LAYER IOs
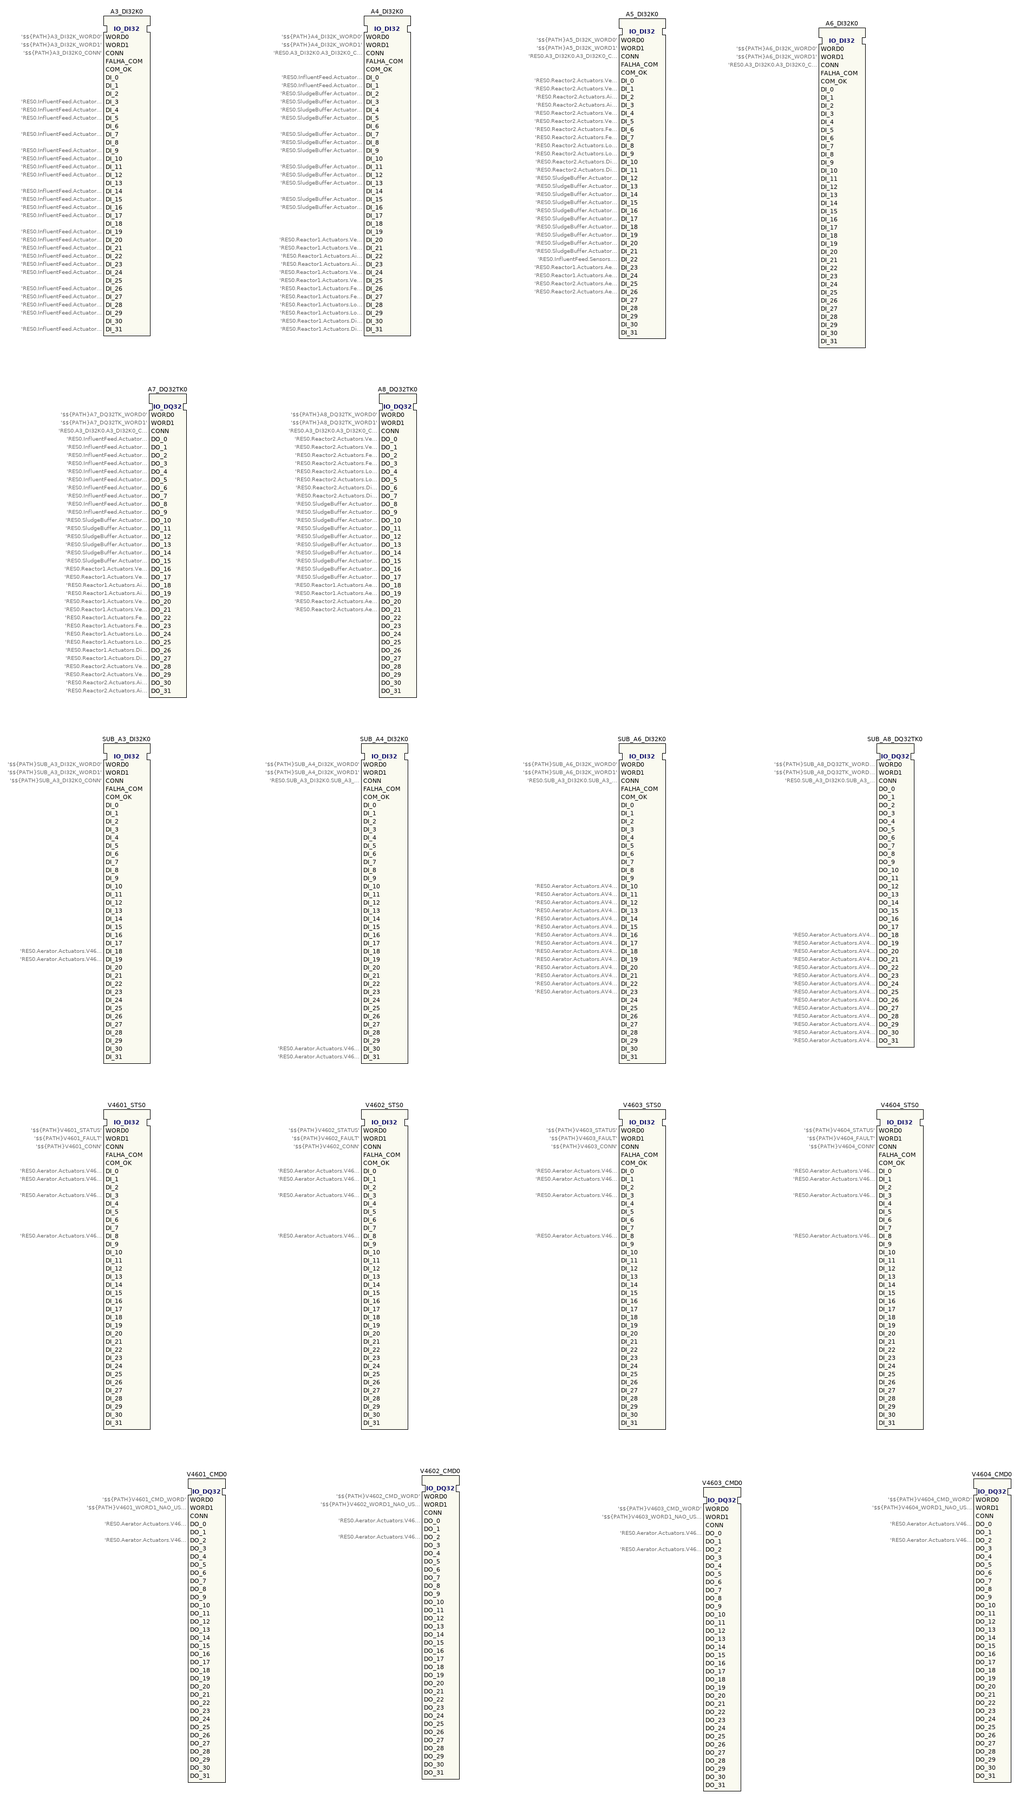
  FBS
    A3_DI32K0 : IO_DI32(WORD0 := '$${PATH}A3_DI32K_WORD0', WORD1 := '$${PATH}A3_DI32K_WORD1', DI_3 := 'RES0.InfluentFeed.Actuators.FeedReactorPump01.LocalPanel.SafetySwitchOff', DI_4 := 'RES0.InfluentFeed.Actuators.FeedReactorPump02.LocalPanel.SafetySwitchOff', DI_5 := 'RES0.InfluentFeed.Actuators.FeedReactorPump03.LocalPanel.SafetySwitchOff', DI_7 := 'RES0.InfluentFeed.Actuators.FeedReactorPump01.LocalPanel.RemoteSelect', DI_9 := 'RES0.InfluentFeed.Actuators.FeedReactorPump01.fbFwd.DIn', DI_10 := 'RES0.InfluentFeed.Actuators.FeedReactorPump01.LocalPanel.ElectricCircuitFail', DI_11 := 'RES0.InfluentFeed.Actuators.FeedReactorPump01.LocalPanel.MoistureDetectionPumpMS', DI_12 := 'RES0.InfluentFeed.Actuators.FeedReactorPump02.LocalPanel.RemoteSelect', DI_14 := 'RES0.InfluentFeed.Actuators.FeedReactorPump02.fbFwd.DIn', DI_15 := 'RES0.InfluentFeed.Actuators.FeedReactorPump02.LocalPanel.ElectricCircuitFail', DI_16 := 'RES0.InfluentFeed.Actuators.FeedReactorPump02.LocalPanel.MoistureDetectionPumpMS', DI_17 := 'RES0.InfluentFeed.Actuators.FeedReactorPump03.LocalPanel.RemoteSelect', DI_19 := 'RES0.InfluentFeed.Actuators.FeedReactorPump03.fbFwd.DIn', DI_20 := 'RES0.InfluentFeed.Actuators.FeedReactorPump03.LocalPanel.ElectricCircuitFail', DI_21 := 'RES0.InfluentFeed.Actuators.FeedReactorPump03.LocalPanel.MoistureDetectionPumpMS', DI_22 := 'RES0.InfluentFeed.Actuators.Mixer01.LocalPanel.PowerFb', DI_23 := 'RES0.InfluentFeed.Actuators.Mixer02.LocalPanel.PowerFb', DI_24 := 'RES0.InfluentFeed.Actuators.Mixer01.LocalPanel.RemoteSelect', DI_26 := 'RES0.InfluentFeed.Actuators.Mixer01.fbFwd.DIn', DI_27 := 'RES0.InfluentFeed.Actuators.Mixer01.LocalPanel.ElectricCircuitFail', DI_28 := 'RES0.InfluentFeed.Actuators.Mixer01.LocalPanel.MoistureDetectionPumpMS', DI_29 := 'RES0.InfluentFeed.Actuators.Mixer02.LocalPanel.RemoteSelect', DI_31 := 'RES0.InfluentFeed.Actuators.Mixer02.fbFwd.DIn', CONN := '$${PATH}A3_DI32K0_CONN');
    A4_DI32K0 : IO_DI32(WORD0 := '$${PATH}A4_DI32K_WORD0', WORD1 := '$${PATH}A4_DI32K_WORD1', DI_0 := 'RES0.InfluentFeed.Actuators.Mixer02.LocalPanel.ElectricCircuitFail', DI_1 := 'RES0.InfluentFeed.Actuators.Mixer02.LocalPanel.MoistureDetectionPumpMS', DI_2 := 'RES0.SludgeBuffer.Actuators.Pump1.LocalPanel.PowerFb', DI_3 := 'RES0.SludgeBuffer.Actuators.Pump2.LocalPanel.PowerFb', DI_4 := 'RES0.SludgeBuffer.Actuators.Pump3.LocalPanel.PowerFb', DI_5 := 'RES0.SludgeBuffer.Actuators.Pump1.LocalPanel.RemoteSelect', DI_7 := 'RES0.SludgeBuffer.Actuators.Pump1.fbFwd.DIn', DI_8 := 'RES0.SludgeBuffer.Actuators.Pump1.LocalPanel.ElectricCircuitFail', DI_9 := 'RES0.SludgeBuffer.Actuators.Pump2.LocalPanel.RemoteSelect', DI_11 := 'RES0.SludgeBuffer.Actuators.Pump2.fbFwd.DIn', DI_12 := 'RES0.SludgeBuffer.Actuators.Pump2.LocalPanel.ElectricCircuitFail', DI_13 := 'RES0.SludgeBuffer.Actuators.Pump3.LocalPanel.RemoteSelect', DI_15 := 'RES0.SludgeBuffer.Actuators.Pump3.fbFwd.DIn', DI_16 := 'RES0.SludgeBuffer.Actuators.Pump3.LocalPanel.ElectricCircuitFail', DI_20 := 'RES0.Reactor1.Actuators.VentAerationGridValve_AV4x107.fbOpen.DIn', DI_21 := 'RES0.Reactor1.Actuators.VentAerationGridValve_AV4x107.fbClose.DIn', DI_22 := 'RES0.Reactor1.Actuators.AirFillValveSludgeDischarge_AV4x171.fbOpen.DIn', DI_23 := 'RES0.Reactor1.Actuators.AirFillValveSludgeDischarge_AV4x171.fbClose.DIn', DI_24 := 'RES0.Reactor1.Actuators.VentSludgeGridValve_AV4x172.fbOpen.DIn', DI_25 := 'RES0.Reactor1.Actuators.VentSludgeGridValve_AV4x172.fbClose.DIn', DI_26 := 'RES0.Reactor1.Actuators.FeedValve_AV4x101.fbOpen.DIn', DI_27 := 'RES0.Reactor1.Actuators.FeedValve_AV4x101.fbClose.DIn', DI_28 := 'RES0.Reactor1.Actuators.LowerLevelValve_AV4x102.fbOpen.DIn', DI_29 := 'RES0.Reactor1.Actuators.LowerLevelValve_AV4x102.fbClose.DIn', DI_30 := 'RES0.Reactor1.Actuators.DischargeValve_AV4x103.fbOpen.DIn', DI_31 := 'RES0.Reactor1.Actuators.DischargeValve_AV4x103.fbClose.DIn', CONN := 'RES0.A3_DI32K0.A3_DI32K0_CONN');
    A5_DI32K0 : IO_DI32(WORD0 := '$${PATH}A5_DI32K_WORD0', WORD1 := '$${PATH}A5_DI32K_WORD1', DI_0 := 'RES0.Reactor2.Actuators.VentAerationGridValve_AV4x107.fbOpen.DIn', DI_1 := 'RES0.Reactor2.Actuators.VentAerationGridValve_AV4x107.fbClose.DIn', DI_2 := 'RES0.Reactor2.Actuators.AirFillValveSludgeDischarge_AV4x171.fbOpen.DIn', DI_3 := 'RES0.Reactor2.Actuators.AirFillValveSludgeDischarge_AV4x171.fbClose.DIn', DI_4 := 'RES0.Reactor2.Actuators.VentSludgeGridValve_AV4x172.fbOpen.DIn', DI_5 := 'RES0.Reactor2.Actuators.VentSludgeGridValve_AV4x172.fbClose.DIn', DI_6 := 'RES0.Reactor2.Actuators.FeedValve_AV4x101.fbOpen.DIn', DI_7 := 'RES0.Reactor2.Actuators.FeedValve_AV4x101.fbClose.DIn', DI_8 := 'RES0.Reactor2.Actuators.LowerLevelValve_AV4x102.fbOpen.DIn', DI_9 := 'RES0.Reactor2.Actuators.LowerLevelValve_AV4x102.fbClose.DIn', DI_10 := 'RES0.Reactor2.Actuators.DischargeValve_AV4x103.fbOpen.DIn', DI_11 := 'RES0.Reactor2.Actuators.DischargeValve_AV4x103.fbClose.DIn', DI_14 := 'RES0.SludgeBuffer.Actuators.ValveBuffer.fbOpen.DIn', DI_15 := 'RES0.SludgeBuffer.Actuators.ValveBuffer.fbClose.DIn', DI_16 := 'RES0.SludgeBuffer.Actuators.ValveInfeed.fbOpen.DIn', DI_17 := 'RES0.SludgeBuffer.Actuators.ValveInfeed.fbClose.DIn', DI_22 := 'RES0.InfluentFeed.Sensors.LevelSwitchInfluentBuffer.pv.DIn', DI_23 := 'RES0.Reactor1.Actuators.AerationBlockValve_AV4x170.fbOpen.DIn', DI_24 := 'RES0.Reactor1.Actuators.AerationBlockValve_AV4x170.fbClose.DIn', DI_25 := 'RES0.Reactor2.Actuators.AerationBlockValve_AV4x170.fbOpen.DIn', DI_26 := 'RES0.Reactor2.Actuators.AerationBlockValve_AV4x170.fbClose.DIn', CONN := 'RES0.A3_DI32K0.A3_DI32K0_CONN', DI_12 := 'RES0.SludgeBuffer.Actuators.ValveSupernatantReturn.fbOpen.DIn', DI_13 := 'RES0.SludgeBuffer.Actuators.ValveSupernatantReturn.fbClose.DIn', DI_18 := 'RES0.SludgeBuffer.Actuators.ValveTank2.fbOpen.DIn', DI_19 := 'RES0.SludgeBuffer.Actuators.ValveTank2.fbClose.DIn', DI_20 := 'RES0.SludgeBuffer.Actuators.ValveTank1.fbOpen.DIn', DI_21 := 'RES0.SludgeBuffer.Actuators.ValveTank1.fbClose.DIn');
    A6_DI32K0 : IO_DI32(WORD0 := '$${PATH}A6_DI32K_WORD0', WORD1 := '$${PATH}A6_DI32K_WORD1', CONN := 'RES0.A3_DI32K0.A3_DI32K0_CONN');
    A7_DQ32TK0 : IO_DQ32(WORD0 := '$${PATH}A7_DQ32TK_WORD0', WORD1 := '$${PATH}A7_DQ32TK_WORD1', DO_0 := 'RES0.InfluentFeed.Actuators.FeedReactorPump01.cmdFwd.DOut', DO_1 := 'RES0.InfluentFeed.Actuators.FeedReactorPump01.LocalPanel.ResetError_ATV', DO_2 := 'RES0.InfluentFeed.Actuators.FeedReactorPump02.cmdFwd.DOut', DO_3 := 'RES0.InfluentFeed.Actuators.FeedReactorPump02.LocalPanel.ResetError_ATV', DO_4 := 'RES0.InfluentFeed.Actuators.FeedReactorPump03.cmdFwd.DOut', DO_5 := 'RES0.InfluentFeed.Actuators.FeedReactorPump03.LocalPanel.ResetError_ATV', DO_6 := 'RES0.InfluentFeed.Actuators.Mixer01.cmdFwd.DOut', DO_7 := 'RES0.InfluentFeed.Actuators.Mixer01.LocalPanel.ResetError_ATV', DO_8 := 'RES0.InfluentFeed.Actuators.Mixer02.cmdFwd.DOut', DO_9 := 'RES0.InfluentFeed.Actuators.Mixer02.LocalPanel.ResetError_ATV', DO_10 := 'RES0.SludgeBuffer.Actuators.Pump1.cmdFwd.DOut', DO_11 := 'RES0.SludgeBuffer.Actuators.Pump1.LocalPanel.ResetError_ATV', DO_12 := 'RES0.SludgeBuffer.Actuators.Pump2.cmdFwd.DOut', DO_13 := 'RES0.SludgeBuffer.Actuators.Pump2.LocalPanel.ResetError_ATV', DO_14 := 'RES0.SludgeBuffer.Actuators.Pump3.cmdFwd.DOut', DO_15 := 'RES0.SludgeBuffer.Actuators.Pump3.LocalPanel.ResetError_ATV', DO_16 := 'RES0.Reactor1.Actuators.VentAerationGridValve_AV4x107.cmdOpen.DOut', DO_17 := 'RES0.Reactor1.Actuators.VentAerationGridValve_AV4x107.cmdClose.DOut', DO_18 := 'RES0.Reactor1.Actuators.AirFillValveSludgeDischarge_AV4x171.cmdOpen.DOut', DO_19 := 'RES0.Reactor1.Actuators.AirFillValveSludgeDischarge_AV4x171.cmdClose.DOut', DO_20 := 'RES0.Reactor1.Actuators.VentSludgeGridValve_AV4x172.cmdOpen.DOut', DO_21 := 'RES0.Reactor1.Actuators.VentSludgeGridValve_AV4x172.cmdClose.DOut', DO_22 := 'RES0.Reactor1.Actuators.FeedValve_AV4x101.cmdOpen.DOut', DO_23 := 'RES0.Reactor1.Actuators.FeedValve_AV4x101.cmdClose.DOut', DO_24 := 'RES0.Reactor1.Actuators.LowerLevelValve_AV4x102.cmdOpen.DOut', DO_25 := 'RES0.Reactor1.Actuators.LowerLevelValve_AV4x102.cmdClose.DOut', DO_26 := 'RES0.Reactor1.Actuators.DischargeValve_AV4x103.cmdOpen.DOut', DO_27 := 'RES0.Reactor1.Actuators.DischargeValve_AV4x103.cmdClose.DOut', DO_28 := 'RES0.Reactor2.Actuators.VentAerationGridValve_AV4x107.cmdOpen.DOut', DO_29 := 'RES0.Reactor2.Actuators.VentAerationGridValve_AV4x107.cmdClose.DOut', DO_30 := 'RES0.Reactor2.Actuators.AirFillValveSludgeDischarge_AV4x171.cmdOpen.DOut', DO_31 := 'RES0.Reactor2.Actuators.AirFillValveSludgeDischarge_AV4x171.cmdClose.DOut', CONN := 'RES0.A3_DI32K0.A3_DI32K0_CONN');
    A8_DQ32TK0 : IO_DQ32(WORD0 := '$${PATH}A8_DQ32TK_WORD0', WORD1 := '$${PATH}A8_DQ32TK_WORD1', DO_0 := 'RES0.Reactor2.Actuators.VentSludgeGridValve_AV4x172.cmdOpen.DOut', DO_1 := 'RES0.Reactor2.Actuators.VentSludgeGridValve_AV4x172.cmdClose.DOut', DO_2 := 'RES0.Reactor2.Actuators.FeedValve_AV4x101.cmdOpen.DOut', DO_3 := 'RES0.Reactor2.Actuators.FeedValve_AV4x101.cmdClose.DOut', DO_4 := 'RES0.Reactor2.Actuators.LowerLevelValve_AV4x102.cmdOpen.DOut', DO_5 := 'RES0.Reactor2.Actuators.LowerLevelValve_AV4x102.cmdClose.DOut', DO_6 := 'RES0.Reactor2.Actuators.DischargeValve_AV4x103.cmdOpen.DOut', DO_7 := 'RES0.Reactor2.Actuators.DischargeValve_AV4x103.cmdClose.DOut', DO_10 := 'RES0.SludgeBuffer.Actuators.ValveBuffer.cmdOpen.DOut', DO_11 := 'RES0.SludgeBuffer.Actuators.ValveBuffer.cmdClose.DOut', DO_12 := 'RES0.SludgeBuffer.Actuators.ValveInfeed.cmdOpen.DOut', DO_13 := 'RES0.SludgeBuffer.Actuators.ValveInfeed.cmdClose.DOut', DO_18 := 'RES0.Reactor1.Actuators.AerationBlockValve_AV4x170.cmdOpen.DOut', DO_19 := 'RES0.Reactor1.Actuators.AerationBlockValve_AV4x170.cmdClose.DOut', DO_20 := 'RES0.Reactor2.Actuators.AerationBlockValve_AV4x170.cmdOpen.DOut', DO_21 := 'RES0.Reactor2.Actuators.AerationBlockValve_AV4x170.cmdClose.DOut', CONN := 'RES0.A3_DI32K0.A3_DI32K0_CONN', DO_8 := 'RES0.SludgeBuffer.Actuators.ValveSupernatantReturn.cmdOpen.DOut', DO_9 := 'RES0.SludgeBuffer.Actuators.ValveSupernatantReturn.cmdClose.DOut', DO_17 := 'RES0.SludgeBuffer.Actuators.ValveTank1.cmdClose.DOut', DO_16 := 'RES0.SludgeBuffer.Actuators.ValveTank1.cmdOpen.DOut', DO_14 := 'RES0.SludgeBuffer.Actuators.ValveTank2.cmdOpen.DOut', DO_15 := 'RES0.SludgeBuffer.Actuators.ValveTank2.cmdClose.DOut');
    SUB_A3_DI32K0 : IO_DI32(WORD0 := '$${PATH}SUB_A3_DI32K_WORD0', WORD1 := '$${PATH}SUB_A3_DI32K_WORD1', DI_18 := 'RES0.Aerator.Actuators.V4603.LocalPanel.PowerFb', DI_19 := 'RES0.Aerator.Actuators.V4604.LocalPanel.PowerFb', CONN := '$${PATH}SUB_A3_DI32K0_CONN');
    SUB_A4_DI32K0 : IO_DI32(WORD0 := '$${PATH}SUB_A4_DI32K_WORD0', WORD1 := '$${PATH}SUB_A4_DI32K_WORD1', DI_30 := 'RES0.Aerator.Actuators.V4601.LocalPanel.PowerFb', DI_31 := 'RES0.Aerator.Actuators.V4602.LocalPanel.PowerFb', CONN := 'RES0.SUB_A3_DI32K0.SUB_A3_DI32K0_CONN');
    SUB_A6_DI32K0 : IO_DI32(WORD0 := '$${PATH}SUB_A6_DI32K_WORD0', WORD1 := '$${PATH}SUB_A6_DI32K_WORD1', DI_10 := 'RES0.Aerator.Actuators.AV46_001.fbOpen.DIn', DI_11 := 'RES0.Aerator.Actuators.AV46_001.fbClose.DIn', DI_12 := 'RES0.Aerator.Actuators.AV46_002.fbOpen.DIn', DI_13 := 'RES0.Aerator.Actuators.AV46_002.fbClose.DIn', DI_14 := 'RES0.Aerator.Actuators.AV46_003.fbOpen.DIn', DI_15 := 'RES0.Aerator.Actuators.AV46_003.fbClose.DIn', DI_16 := 'RES0.Aerator.Actuators.AV46_012.fbOpen.DIn', DI_17 := 'RES0.Aerator.Actuators.AV46_012.fbClose.DIn', DI_18 := 'RES0.Aerator.Actuators.AV46_022.fbOpen.DIn', DI_19 := 'RES0.Aerator.Actuators.AV46_022.fbClose.DIn', DI_20 := 'RES0.Aerator.Actuators.AV46_032.fbOpen.DIn', DI_21 := 'RES0.Aerator.Actuators.AV46_032.fbClose.DIn', DI_22 := 'RES0.Aerator.Actuators.AV46_042.fbOpen.DIn', DI_23 := 'RES0.Aerator.Actuators.AV46_042.fbClose.DIn', CONN := 'RES0.SUB_A3_DI32K0.SUB_A3_DI32K0_CONN');
    SUB_A8_DQ32TK0 : IO_DQ32(WORD0 := '$${PATH}SUB_A8_DQ32TK_WORD0', WORD1 := '$${PATH}SUB_A8_DQ32TK_WORD1', DO_18 := 'RES0.Aerator.Actuators.AV46_001.cmdOpen.DOut', DO_19 := 'RES0.Aerator.Actuators.AV46_001.cmdClose.DOut', DO_20 := 'RES0.Aerator.Actuators.AV46_002.cmdOpen.DOut', DO_21 := 'RES0.Aerator.Actuators.AV46_002.cmdClose.DOut', DO_22 := 'RES0.Aerator.Actuators.AV46_003.cmdOpen.DOut', DO_23 := 'RES0.Aerator.Actuators.AV46_003.cmdClose.DOut', DO_24 := 'RES0.Aerator.Actuators.AV46_012.cmdOpen.DOut', DO_25 := 'RES0.Aerator.Actuators.AV46_012.cmdClose.DOut', DO_26 := 'RES0.Aerator.Actuators.AV46_022.cmdOpen.DOut', DO_27 := 'RES0.Aerator.Actuators.AV46_022.cmdClose.DOut', DO_28 := 'RES0.Aerator.Actuators.AV46_032.cmdOpen.DOut', DO_29 := 'RES0.Aerator.Actuators.AV46_032.cmdClose.DOut', DO_30 := 'RES0.Aerator.Actuators.AV46_042.cmdOpen.DOut', DO_31 := 'RES0.Aerator.Actuators.AV46_042.cmdClose.DOut', CONN := 'RES0.SUB_A3_DI32K0.SUB_A3_DI32K0_CONN');
    V4601_STS0 : IO_DI32(WORD0 := '$${PATH}V4601_STATUS', WORD1 := '$${PATH}V4601_FAULT', CONN := '$${PATH}V4601_CONN', DI_0 := 'RES0.Aerator.Actuators.V4601.LocalPanel.RemoteSelect', DI_1 := 'RES0.Aerator.Actuators.V4601.fbFwd.DIn', DI_3 := 'RES0.Aerator.Actuators.V4601.LocalPanel.FrequencyInverterFail', DI_8 := 'RES0.Aerator.Actuators.V4601.LocalPanel.AtvReady');
    V4601_CMD0 : IO_DQ32(WORD0 := '$${PATH}V4601_CMD_WORD', WORD1 := '$${PATH}V4601_WORD1_NAO_USADA', DO_0 := 'RES0.Aerator.Actuators.V4601.cmdFwd.DOut', DO_2 := 'RES0.Aerator.Actuators.V4601.LocalPanel.ResetError_ATV');
    V4602_STS0 : IO_DI32(WORD0 := '$${PATH}V4602_STATUS', WORD1 := '$${PATH}V4602_FAULT', CONN := '$${PATH}V4602_CONN', DI_0 := 'RES0.Aerator.Actuators.V4602.LocalPanel.RemoteSelect', DI_1 := 'RES0.Aerator.Actuators.V4602.fbFwd.DIn', DI_3 := 'RES0.Aerator.Actuators.V4602.LocalPanel.FrequencyInverterFail', DI_8 := 'RES0.Aerator.Actuators.V4602.LocalPanel.AtvReady');
    V4602_CMD0 : IO_DQ32(WORD0 := '$${PATH}V4602_CMD_WORD', WORD1 := '$${PATH}V4602_WORD1_NAO_USADA', DO_0 := 'RES0.Aerator.Actuators.V4602.cmdFwd.DOut', DO_2 := 'RES0.Aerator.Actuators.V4602.LocalPanel.ResetError_ATV');
    V4603_STS0 : IO_DI32(WORD0 := '$${PATH}V4603_STATUS', WORD1 := '$${PATH}V4603_FAULT', CONN := '$${PATH}V4603_CONN', DI_0 := 'RES0.Aerator.Actuators.V4603.LocalPanel.RemoteSelect', DI_1 := 'RES0.Aerator.Actuators.V4603.fbFwd.DIn', DI_3 := 'RES0.Aerator.Actuators.V4603.LocalPanel.FrequencyInverterFail', DI_8 := 'RES0.Aerator.Actuators.V4603.LocalPanel.AtvReady');
    V4603_CMD0 : IO_DQ32(WORD0 := '$${PATH}V4603_CMD_WORD', WORD1 := '$${PATH}V4603_WORD1_NAO_USADA', DO_0 := 'RES0.Aerator.Actuators.V4603.cmdFwd.DOut', DO_2 := 'RES0.Aerator.Actuators.V4603.LocalPanel.ResetError_ATV');
    V4604_STS0 : IO_DI32(WORD0 := '$${PATH}V4604_STATUS', WORD1 := '$${PATH}V4604_FAULT', CONN := '$${PATH}V4604_CONN', DI_0 := 'RES0.Aerator.Actuators.V4604.LocalPanel.RemoteSelect', DI_1 := 'RES0.Aerator.Actuators.V4604.fbFwd.DIn', DI_3 := 'RES0.Aerator.Actuators.V4604.LocalPanel.FrequencyInverterFail', DI_8 := 'RES0.Aerator.Actuators.V4604.LocalPanel.AtvReady');
    V4604_CMD0 : IO_DQ32(WORD0 := '$${PATH}V4604_CMD_WORD', WORD1 := '$${PATH}V4604_WORD1_NAO_USADA', DO_0 := 'RES0.Aerator.Actuators.V4604.cmdFwd.DOut', DO_2 := 'RES0.Aerator.Actuators.V4604.LocalPanel.ResetError_ATV');
  END_FBS
END_LAYER
